TYPE ST_XYPos :
STRUCT
	X			:LREAL;
	Y			:LREAL;
END_STRUCT
END_TYPE

(* stored: Version 1.1.0.1, ProductVersion 3.1.4024.12
   DUT ST_XYPos: Id {79d14705-9756-4439-9490-3f7da75b58bd} *)
